FUNCTION IncUDINT : UDINT		// Increments the given UINT value
VAR_IN_OUT
	ioNum:	UDINT;		// Value to increment
END_VAR

IncUDINT := ioNum := ioNum + 1;

END_FUNCTION

(* stored: Version 1.1.0.1, ProductVersion 3.1.4026.18
   POU IncUDINT: Id {d1295a8b-3754-4a8c-87df-265ebfe748cc}, SpecialFunc None *)
